PROGRAM Logowanie
VAR
	
	pClient                : POINTER TO VisuElems.VisuStructClientData;
	wsCurrentUser			: WSTRING;
END_VAR

//pClient := VisuElems.g_ClientManager.GetNextClient(); 
wsCurrentUser:=VisuElemsWinControls.CurrentUserName;
//IF wsCurrentUser<>"admin" AND GVL_HMI.hmiPanel.uiMenu=5  THEN
	//VisuUserManagement.OpenLoginDialog(pClient);
//END_IF

END_PROGRAM

(* stored: Version 1.1.0.1, ProductVersion 3.1.4024.3
   POU Logowanie: Id {22b85a99-3ad8-4c79-b7a2-79474d78307b}, SpecialFunc None *)
